// TIA Portal V19 export
FUNCTION_BLOCK "TYPIC_C106_BF_HSI"   // FB85, FBD
TITLE = TYPIC_C106_BF_HSI: Hoogspanningsinstallatie
{ S7_Optimized_Access := 'TRUE' }
AUTHOR : OCOTECH
FAMILY : Typical
NAME : C106.801
// Logisch Object Besturing: C106.801
// 
// Het doel van de BF HSI (hoogspanningsinstallatie) is om de algemene opvolging te voorzien van de hoogspanningsinstallatie.
// stored: MemoryReserve 10, SetENOAutomatically false
   VAR_INPUT
      STU_ALG_LCK_SIG { ExternalAccessible := 'False'; ExternalVisible := 'False'; ExternalWritable := 'False'} : USInt;   // Onderdruk alarmen
   END_VAR
   VAR_OUTPUT
      AUT_STS_HSI { ExternalAccessible := 'False'; ExternalVisible := 'False'; ExternalWritable := 'False'} : Array[0..1] of Bool;   // Standmelding van de vermogenschakelaar van de hoogspanning, naar de coordinerende functie Energiemonitor
   END_VAR
   VAR_IN_OUT
      VAR_IF_HSI : "C106_VAR_IF_HSI_TYPIC";   // Struct met alle variabelen van de interne besturing van de hoogspanningsinstallatie en de status van de hoogspanningslus
      VAR_REL : Array[*] of "C106_VAR_REL_TYPIC";   // Array met de standmelding van alle vermogenschakelaars (gekoppeld aan het beveiligingsrelais)
   END_VAR
   VAR
      SIG { ExternalWritable := 'False'} : Struct   // Signaleringen
         AB01 : Bool;   // Hoogspanningsinstallatie niet beschikbaar
         AB02 : Bool;   // Hoogspanningsinstallatie beperkt beschikbaar
         AA01 : Bool;   // Hoogspanningsinstallatie niet observeerbaar
         AA02 : Bool;   // Hoogspanningsinstallatie storing algemeen
         A001 : Bool;   // Beveiliging aangesproken
         A002 : Bool;   // Hoogspanningsinstallatie in storing
         A003 : Bool;   // Algemene storing hoogspanningsinstallatie
         A004 : Bool;   // Hoogspanningslus is geopend
      END_STRUCT;
      VAR { ExternalWritable := 'False'} : Struct   // Variabelen
         LUS_STS : USInt;   // Status van de hoogspanningslus
         BSC : USInt;   // Geeft de beschikbaarheid van de hoogspanningsinstallatie aan
         VGV_SIG_VOP : Bool;   // TRUE = Signaleringen vrijgegeven voor verkeersoperator FALSE = Onderdrukt
      END_STRUCT;
   END_VAR
BEGIN

REGION Network 1: START
END_REGION

REGION Network 2: +++ Verwerking meetwaarden en statussen +++
   // Verwerken van de ontvangen meetwaarden en statussen
END_REGION

REGION Network 3: +++ Bepalen werkingsregime hoogspanningsinstallatie +++
   // Het bepalen van het werkingsregime van de hoogspanningsinstallatie in samenspraak met de noodstroominstallatie
END_REGION

REGION Network 4: +++ Bepalen status hoogspanningslus +++
   // De status van de hoogspanningslus geeft aan of de hoogspanningslus onderbroken is of niet
END_REGION

REGION Network 5: +++ Doorkoppelen gegevens vermogen en energie naar coördinerende functie energiemonitoring +++
   // De actuele vermogen en energiemeting wordt doorgegeven aan de coordinerende functie Energievoorziening.
END_REGION

REGION Network 6: +++ Doorkoppelen status vermogenschakelaars HSI naar coördinerende functie energiemonitoring +++
   // De status van de vermogenschakelaars van de hoogspanningsinstallatie wordt doorgegeven aan de coordinerende functie Energievoorziening
END_REGION

REGION Network 7: +++ Bepalen beschikbaarheidsstatus +++
   // Beschikbaarheidsstatus (beschikbaar / beperkt beschikbaar / niet beschikbaar) bepalen.
END_REGION

REGION Network 8 (SCL): Beschikbaarheidsstatus bepalen
   IF 
       //voorwaarden "Niet beschikbaar"
       TRUE
   THEN
       //Beschikbaarheidsstatus = Niet Beschikbaar
       #VAR.BSC:= "NietBeschikbaar";
   ELSIF
       //voorwaarden "Beperkt beschikbaar"
       TRUE
   THEN
       //Beschikbaarheidsstatus = Beperkt Beschikbaar
       #VAR.BSC:= "Beperkt";
   ELSE
       //Beschikbaarheidsstatus = Beschikbaar
       #VAR.BSC:= "Beschikbaar";
   END_IF;
END_REGION

REGION Network 9: +++ Signaleringen +++
   // Aanmaken signaleringen
END_REGION

REGION Network 10 (SCL): Signaleringen voor de onderhoudsoperator
   // Signalering van de storingen ontvangen vanuit de interne sturing
   #SIG.A001 := #VAR_IF_HSI.STO.A001;
   #SIG.A002 := #VAR_IF_HSI.STO.A002;
   #SIG.A003 := #VAR_IF_HSI.STO.A003;
   #SIG.A004 := #VAR_IF_HSI.STO.A004;
END_REGION

REGION Network 11: Signalering AB01 : Niet Beschikbaar
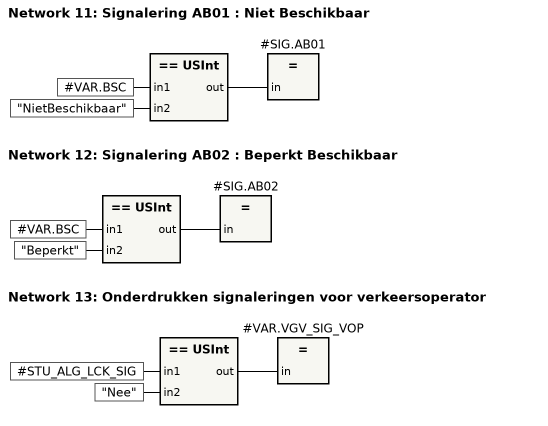
   #SIG.AB01 := #VAR.BSC = "NietBeschikbaar";
END_REGION

REGION Network 12: Signalering AB02 : Beperkt Beschikbaar
   #SIG.AB02 := #VAR.BSC = "Beperkt";
END_REGION

REGION Network 13: Onderdrukken signaleringen voor verkeersoperator
   // Via de variabele VGV_SIG_VOP wordt aan IRIS SCADA doorgegeven of signaleringen (bestemd voor de verkeersoperator) van de deze functie zichtbaar (of onderdrukt) moeten zijn.
   #VAR.VGV_SIG_VOP := #STU_ALG_LCK_SIG = "Nee";
END_REGION

REGION Network 14: EINDE
   // Variabelen van intern scada rakvlak naar outputs copieren
END_REGION
END_FUNCTION_BLOCK
